FUNCTION_BLOCK FB_CSV_RobotDataWriter
VAR_INPUT
	bWriteLine:	BOOL;
	sFileName:	STRING;
	stRobotData : ST_UR;
	bEnable : BOOL;
END_VAR
VAR_OUTPUT
	bBusy:	BOOL;
	bFileOpen : BOOL;
	bError:	BOOL;
	sError:	STRING;
END_VAR
VAR
	fbFileOpen:	FB_FileOpen;
	fbFilePuts:	FB_FilePuts;
	fbFileClose:	FB_FileClose;
	
	rtWrite:	R_TRIG;
	
	nState:	INT;
	sTempPathName:	STRING;
	sDataString1:	STRING(255);
	sDataString2:	STRING(255);
	
	nLastTimestamp : LWORD;
END_VAR

//rtWrite(	CLK := bWriteLine);

CASE nState OF
	0:	(*IDLE*)
		bBusy := FALSE;
		// choose state		
		IF bFileOpen AND NOT bEnable THEN
			// close file
			nState := 30;
		END_IF
		
		IF nLastTimestamp <> stRobotData.RobotModeData.Timestamp THEN
			bWriteLine := FALSE;
			bBusy := TRUE;
			bError := FALSE;
			sError := '';
			sTempPathName := CONCAT(CONCAT('D:\PLCTempData\',sFileName),'.csv');
			// Build Datastrings
			// uint = 20 characters, word = 6 characters, bool = 5 characters, lword = 11, lreal = 16/15 
			// 12 ulints = 240 bytes max string length of 255
			sDataString1 := '';
			//time
			sDataString1 := INSERT(sDataString1,CONCAT(LWORD_TO_STRING(Global.nCurrentTime),','),LEN(sDataString1));
			sDataString1 := INSERT(sDataString1,CONCAT(LWORD_TO_STRING(stRobotData.RobotModeData.Timestamp),','),LEN(sDataString1));
			//position
			sDataString1 := INSERT(sDataString1,CONCAT(LREAL_TO_STRING(stRobotData.JointData.j1_qactual),','),LEN(sDataString1));
			sDataString1 := INSERT(sDataString1,CONCAT(LREAL_TO_STRING(stRobotData.JointData.j2_qactual),','),LEN(sDataString1));
			sDataString1 := INSERT(sDataString1,CONCAT(LREAL_TO_STRING(stRobotData.JointData.j3_qactual),','),LEN(sDataString1));
			sDataString1 := INSERT(sDataString1,CONCAT(LREAL_TO_STRING(stRobotData.JointData.j4_qactual),','),LEN(sDataString1));
			sDataString1 := INSERT(sDataString1,CONCAT(LREAL_TO_STRING(stRobotData.JointData.j5_qactual),','),LEN(sDataString1));
			sDataString1 := INSERT(sDataString1,CONCAT(LREAL_TO_STRING(stRobotData.JointData.j6_qactual),','),LEN(sDataString1));
			
			// Second half of part data
			sDataString2 := '';
			//velocity
			sDataString2 := INSERT(sDataString2,CONCAT(LREAL_TO_STRING(stRobotData.JointData.j1_qdactual),','),LEN(sDataString2));
			sDataString2 := INSERT(sDataString2,CONCAT(LREAL_TO_STRING(stRobotData.JointData.j2_qdactual),','),LEN(sDataString2));
			sDataString2 := INSERT(sDataString2,CONCAT(LREAL_TO_STRING(stRobotData.JointData.j3_qdactual),','),LEN(sDataString2));
			sDataString2 := INSERT(sDataString2,CONCAT(LREAL_TO_STRING(stRobotData.JointData.j4_qdactual),','),LEN(sDataString2));
			sDataString2 := INSERT(sDataString2,CONCAT(LREAL_TO_STRING(stRobotData.JointData.j5_qdactual),','),LEN(sDataString2));
			sDataString2 := INSERT(sDataString2,CONCAT(LREAL_TO_STRING(stRobotData.JointData.j6_qdactual),','),LEN(sDataString2));
			// Tool XYZ
			sDataString2 := INSERT(sDataString2,CONCAT(LREAL_TO_STRING(stRobotData.CartesianInfo.ToolX),','),LEN(sDataString2));
			sDataString2 := INSERT(sDataString2,CONCAT(LREAL_TO_STRING(stRobotData.CartesianInfo.ToolY),','),LEN(sDataString2));
			sDataString2 := INSERT(sDataString2,CONCAT(LREAL_TO_STRING(stRobotData.CartesianInfo.ToolZ),','),LEN(sDataString2));
			// New line
			sDataString2 := CONCAT(sDataString2,'$N');
			
			// Keep track of new messages
			nLastTimestamp := stRobotData.RobotModeData.Timestamp;
			
			// go to next state
			IF bFileOpen THEN
				// start writing strings
				nState := 20;
			ELSE
				// open file
				nState := 10;
			END_IF
		END_IF		
	
	10:	(*Open File*)	
		fbFileOpen(	sPathName := sTempPathName,
					nMode := FOPEN_MODEAPPEND,
					bExecute := TRUE,
					tTimeOut := T#1S);
		IF NOT fbFileOpen.bBusy THEN
			fbFileOpen(	bExecute := FALSE);
			IF fbFileOpen.bError THEN
				bError := TRUE;
				sError := 'Could Not Open File';
				nState := 0;
			ELSE
				bFileOpen := TRUE;
				nState := nState + 10;
			END_IF
		END_IF
		
	20:	(*Write Line To File*)
		fbFilePuts(	hFile := fbFileOpen.hFile,
					sLine := sDataString1,
					bExecute := TRUE,
					tTimeout := T#1S);
		IF NOT fbFilePuts.bBusy THEN
			fbFilePuts(	bExecute := FALSE);
			IF fbFilePuts.bError THEN
				bError := TRUE;
				sError := 'Could not write to file';
				nState := nState + 10;
			ELSE
				nState := nState + 1;
			END_IF
		END_IF
	21:	(*Write Line To File*)
		fbFilePuts(	hFile := fbFileOpen.hFile,
					sLine := sDataString2,
					bExecute := TRUE,
					tTimeout := T#1S);
		IF NOT fbFilePuts.bBusy THEN
			fbFilePuts(	bExecute := FALSE);
			IF fbFilePuts.bError THEN
				bError := TRUE;
				sError := 'Could not write to file';
				nState := 30;
			ELSE
				IF bEnable THEN
					nState := 0;
				ELSE
					nState := 30;
				END_IF
			END_IF
		END_IF
		
	30:	(*Close File*)
		fbFileClose(	hFile := fbFileOpen.hFile,
						bExecute := TRUE,
						tTimeout := T#1S);
		IF NOT fbFileClose.bBusy THEN
			fbFileClose(	bExecute := FALSE);
			IF fbFileClose.bError THEN
				bError := TRUE;
				sError := 'Could not close file';
				nState := 0;
			ELSE
				bFileOpen := FALSE;
				nState := 0;
			END_IF
		END_IF
END_CASE

END_FUNCTION_BLOCK

(* stored: Version 1.1.0.1, ProductVersion 3.1.4020.12
   POU FB_CSV_RobotDataWriter: Id {a29298f2-3bdb-4037-8347-98339629e162}, SpecialFunc None *)
